{attribute 'linkalways'} 
{attribute 'no_explicit_call' := 'This FB is a CLASS and must be accessed using methods or properties'}
{attribute 'enable_dynamic_creation'}
FUNCTION_BLOCK _TIME_OF_DAY EXTENDS DatatypeBase
VAR
	localData : TIME_OF_DAY;
	activeData : REFERENCE TO TIME_OF_DAY REF= localData;
END_VAR

PROPERTY PUBLIC Address : PVOID
GET
Address := ADR(activeData);
END_GET
END_PROPERTY

METHOD PUBLIC ClearReference
VAR_INPUT
END_VAR
activeData REF= localData;
END_METHOD

METHOD PUBLIC Clone : I_Datatype
VAR
    pClone : POINTER TO _TIME_OF_DAY;
END_VAR
pClone := __NEW(_TIME_OF_DAY(InitialValue := Value));
Clone := pClone^;
END_METHOD

METHOD FB_init : BOOL
VAR_INPUT
	bInitRetains : BOOL; // if TRUE, the retain variables are initialized (warm start / cold start)
	bInCopyCode : BOOL;  // if TRUE, the instance afterwards gets moved WORDo the copy code (online change)
	InitialValue : TIME_OF_DAY;
END_VAR
localData := InitialValue;
END_METHOD

METHOD PUBLIC MakeReferenceTo
VAR_INPUT
	ReferenceTarget : REFERENCE TO TIME_OF_DAY;
END_VAR
activeData REF= ReferenceTarget;
END_METHOD

METHOD PUBLIC SerializeWith
VAR_INPUT
	Serializer : I_Serializer;
END_VAR
Serializer.AddTod(activeData);
END_METHOD

PROPERTY PUBLIC Size : UDINT
GET
Size := SIZEOF(activeData);
END_GET
END_PROPERTY

METHOD TryDeserializeFrom : BOOL
VAR_INPUT
	Deserializer : I_Deserializer;
	Feedback : I_DeserializerFeedback;
END_VAR
TryDeserializeFrom := Deserializer.TryGetTod(activeData, Feedback);
END_METHOD

METHOD TryMakeReferenceTo : BOOL
VAR_INPUT
	Target : I_Datatype;
END_VAR
VAR
	pTargetData : POINTER TO TIME_OF_DAY;
END_VAR
IF NOT (Target.TypeName = TypeName) THEN
	RETURN;
END_IF

pTargetData := Target.Address;
activeData REF= pTargetData^;
TryMakeReferenceTo := TRUE;
END_METHOD

PROPERTY PUBLIC TypeName : T_MAXSTRING
GET
TypeName := 'TIME_OF_DAY';
END_GET
END_PROPERTY

PROPERTY PUBLIC Value : TIME_OF_DAY
GET
Value := activeData;
END_GET
SET
activeData := Value;
END_SET
END_PROPERTY

END_FUNCTION_BLOCK

(* stored: Version 1.1.0.1, ProductVersion 3.1.4024.12
   POU _TIME_OF_DAY: Id {09091076-4c50-0c79-075a-93b2440ef830}, SpecialFunc None
   Folder Constructor: Id {bc75c500-de81-095c-1afc-f7b783e9397d}
   Property Address: Id {971a8994-f5cd-0ee9-1115-61454c7df407}
   Get Get: Id {43b22550-8ac9-0820-04b3-3f4bf07a2383}
   Method ClearReference: Id {e729ce88-b9ea-032f-3f2d-6bc83fd21c56}
   Method Clone: Id {8889ee8d-d9d4-0a6f-16dc-aae4357a9077}
   Method FB_init: Id {5dbe585a-3e5b-02a1-199a-3e99a46aa38d}
   Method MakeReferenceTo: Id {ce3da2d1-083a-01c5-3259-bad5bf7dad39}
   Method SerializeWith: Id {704258f6-87eb-0ab3-07c4-104ee2283e18}
   Property Size: Id {3e1f3b9e-d588-014b-2dd2-caab1fc808fe}
   Get Get: Id {fcab8b16-d06b-0978-21b1-1306d8d23688}
   Method TryDeserializeFrom: Id {aa41599a-0230-0d11-2bdc-8596be3bd35a}
   Method TryMakeReferenceTo: Id {657a6ad8-8b41-0476-1761-edb8be0a3f66}
   Property TypeName: Id {df89fd02-abc2-023d-29d4-0197a773c90a}
   Get Get: Id {f75f0d69-8b55-0f23-28a0-425f2700783a}
   Property Value: Id {60d8e0d8-8150-032e-240f-cd363f409430}
   Get Get: Id {6c04b15d-2448-0530-175a-0c6bc9b7cc91}
   Set Set: Id {c624266e-72ec-0200-1751-4077690ac1b4} *)
